# EPICS autosave request: 3-3/GalilSup/Db/galil_forward_transform.req
#Forward transform equation
$(P)$(M)_FTRANSFORM_SP.VAL
$(P)$(M)_FTRANSFORM_SP.DESC
